(* IEC 61131-3 sources: repolevel_ST_code_completion/output/0127完整版本_带planner/repoeval_ProductionLine/readful_result_no_provide, 6 files *)

(* ---- Motor.st ---- *)
VAR
	WaitTimer: TON;
	InternalSequenceDelay: TIME;
END_VAR

IF MotorI.liga THEN
	TurnOn();
END_IF;

IF MotorI.desliga THEN
	TurnOff();
END_IF;

IF MotorI.settime THEN
	SetWaitTime(SequenceDelay := MotorI.timetemp);
END_IF;

IF MotorI.setfault THEN
	SetFault();
END_IF;

IF MotorI.reset THEN
	MotorO.FaultStatus := FALSE;
	WaitTimer(IN := FALSE);
END_IF;
END_FUNCTION_BLOCK

(* ---- Motor_ResetFault.st ---- *)
VAR
	ResetDetect: R_TRIG;
	ResetSuccessful: BOOL;
END_VAR

ResetDetect(CLK := MotorI.ResetSignal);

IF ResetDetect.Q THEN
	MotorO.FaultStatus := FALSE;
	MotorO.OperationStatus := READY; // Assuming READY is the default operation status
	ResetSuccessful := TRUE;
ELSE
	ResetSuccessful := FALSE;
END_IF;

ResetFault := ResetSuccessful;
RETURN;
END_OTHER

(* ---- Motor_SetFault.st ---- *)
VAR
	OverloadDetected: BOOL;
END_VAR

OverloadDetected := MotorI.Overload;

IF OverloadDetected THEN
	MotorO.FaultStatus := TRUE;
	MotorO.Coil := FALSE; // Turn off the motor
	SetFault := TRUE; // Fault successfully handled
ELSE
	SetFault := FALSE; // No fault detected
END_IF;
END_OTHER

(* ---- Motor_SetWaitTime.st ---- *)
VAR
	IsValidDelay: BOOL;
END_VAR

// Step 1: Check if SequenceDelay is a valid time value (non-negative)
IsValidDelay := SequenceDelay >= T#0ms;

// Step 2: Update MotorI.WaitTime if SequenceDelay is valid
IF IsValidDelay THEN
	MotorI.WaitTime := SequenceDelay;
END_IF;

// Step 3: Copy updated MotorI to MotorO
MotorO := MotorI;

// Step 4: Return success flag
RETURN TRUE;
END_OTHER

(* ---- Motor_TurnOff.st ---- *)
VAR
	OperationSuccessful: BOOL;
END_VAR

OperationSuccessful := FALSE;

IF MotorI.AllowTurnOff THEN
	MotorO.Coil := FALSE;
	MotorO.Status := 'Off';
	OperationSuccessful := TRUE;
END_IF;

TurnOff := OperationSuccessful;
RETURN;
END_OTHER

(* ---- Motor_TurnOn.st ---- *)
VAR
	WaitTimer: TON;
END_VAR

IF MotorI.FaultStatus THEN
	RETURN := FALSE;
	RETURN;
END_IF;

WaitTimer(IN := TRUE, PT := MotorI.DelayTime);

IF NOT WaitTimer.Q THEN
	RETURN := FALSE;
	RETURN;
END_IF;

MotorO.Coil := TRUE;
RETURN := TRUE;
END_OTHER
